FUNCTION_BLOCK FB_WP_Ablaufsteuerung
VAR_IN_OUT
	Zustand			: ST_WP_Zustand;
	Stellwert		: ST_WP_Stellwert;
END_VAR
VAR_INPUT
	Steuerung		: ST_WP_Steuerung;
	Parameter		: ST_WP_Parameter;
END_VAR
VAR_OUTPUT
END_VAR
VAR
	Timer			: TON;
END_VAR

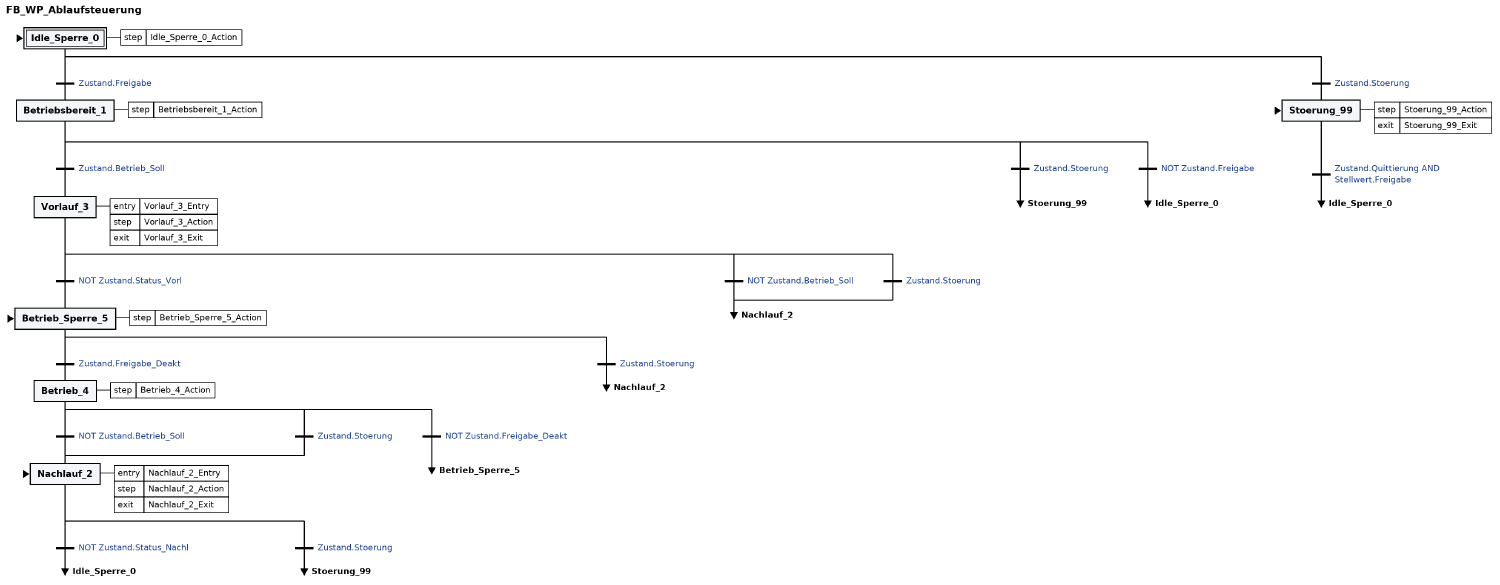
INITIAL_STEP Idle_Sperre_0:
    Idle_Sperre_0_Action(N);  // step action
END_STEP
TRANSITION FROM Idle_Sperre_0 TO Betriebsbereit_1
    := Zustand.Freigabe;
END_TRANSITION
TRANSITION FROM Idle_Sperre_0 TO Stoerung_99
    := Zustand.Stoerung;
END_TRANSITION
STEP Stoerung_99:
    Stoerung_99_Action(N);  // step action
    Stoerung_99_Exit(P0);  // exit action
END_STEP
TRANSITION FROM Stoerung_99 TO Idle_Sperre_0
    := Zustand.Quittierung AND Stellwert.Freigabe;
END_TRANSITION
STEP Betriebsbereit_1:
    Betriebsbereit_1_Action(N);  // step action
END_STEP
TRANSITION FROM Betriebsbereit_1 TO Vorlauf_3
    := Zustand.Betrieb_Soll;
END_TRANSITION
TRANSITION FROM Betriebsbereit_1 TO Stoerung_99
    := Zustand.Stoerung;
END_TRANSITION
TRANSITION FROM Betriebsbereit_1 TO Idle_Sperre_0
    := NOT Zustand.Freigabe;
END_TRANSITION
STEP Vorlauf_3:
    Vorlauf_3_Entry(P1);  // entry action
    Vorlauf_3_Action(N);  // step action
    Vorlauf_3_Exit(P0);  // exit action
END_STEP
TRANSITION FROM Vorlauf_3 TO Betrieb_Sperre_5
    := NOT Zustand.Status_Vorl;
END_TRANSITION
TRANSITION FROM Vorlauf_3 TO Nachlauf_2
    := NOT Zustand.Betrieb_Soll;
END_TRANSITION
TRANSITION FROM Vorlauf_3 TO Nachlauf_2
    := Zustand.Stoerung;
END_TRANSITION
STEP Betrieb_Sperre_5:
    Betrieb_Sperre_5_Action(N);  // step action
END_STEP
TRANSITION FROM Betrieb_Sperre_5 TO Betrieb_4
    := Zustand.Freigabe_Deakt;
END_TRANSITION
TRANSITION FROM Betrieb_Sperre_5 TO Nachlauf_2
    := Zustand.Stoerung;
END_TRANSITION
STEP Betrieb_4:
    Betrieb_4_Action(N);  // step action
END_STEP
TRANSITION FROM Betrieb_4 TO Nachlauf_2
    := NOT Zustand.Betrieb_Soll;
END_TRANSITION
TRANSITION FROM Betrieb_4 TO Nachlauf_2
    := Zustand.Stoerung;
END_TRANSITION
TRANSITION FROM Betrieb_4 TO Betrieb_Sperre_5
    := NOT Zustand.Freigabe_Deakt;
END_TRANSITION
STEP Nachlauf_2:
    Nachlauf_2_Entry(P1);  // entry action
    Nachlauf_2_Action(N);  // step action
    Nachlauf_2_Exit(P0);  // exit action
END_STEP
TRANSITION FROM Nachlauf_2 TO Idle_Sperre_0
    := NOT Zustand.Status_Nachl;
END_TRANSITION
TRANSITION FROM Nachlauf_2 TO Stoerung_99
    := Zustand.Stoerung;
END_TRANSITION

ACTION Betrieb_4_Action:
(* Stellwert setzen *)
Stellwert.Betrieb := TRUE;

(* Zustand setzen *)
Zustand.Status := E_WP_Zustand_Status_Betrieb;
END_ACTION

ACTION Betrieb_Sperre_5_Action:
(* Stellwert setzen *)
Stellwert.Betrieb := TRUE;

(* Zustand setzen *)
Zustand.Status := E_WP_Zustand_Status_Betrieb_Sperre;
END_ACTION

ACTION Betriebsbereit_1_Action:
(* Stellwert setzen *)
Stellwert.Betrieb := FALSE;
Stellwert.Freigabe := TRUE;

(* Zustand setzen *)
Zustand.Status := E_WP_Zustand_Status_Betriebsbereit;
END_ACTION

ACTION Idle_Sperre_0_Action:
(* Stellwert setzen *)
Stellwert.Betrieb := FALSE;

(* Zustand setzen *)
Zustand.Status := E_WP_Zustand_Status_Idle_Sperre;
END_ACTION

ACTION Nachlauf_2_Action:
(* Nachlauf Timer starten *)
Timer( 	IN := Zustand.Status_Nachl,
		PT := DINT_TO_TIME(Parameter.Zeit_Nachl)
);
Zustand.Status_Nachl	:= NOT(Timer.Q AND NOT Zustand.Betrieb);

(* Stellwert setzen *)
Stellwert.Betrieb := FALSE;
Stellwert.Freigabe := FALSE;

(* Zustand setzen *)
Zustand.Status := E_WP_Zustand_Status_Nachl;
END_ACTION

ACTION Nachlauf_2_Entry:
Zustand.Status_Nachl := TRUE;
(* Reset Timer *)
Timer(IN := FALSE);
END_ACTION

ACTION Nachlauf_2_Exit:
Zustand.Status_Nachl := FALSE;
END_ACTION

ACTION Stoerung_99_Action:
(* Stellwert setzen *)
Stellwert.Betrieb := FALSE;

(* Zustand setzen *)
Zustand.Stoerung := TRUE;
Zustand.Status := E_WP_Zustand_Status_Stoerung;
END_ACTION

ACTION Stoerung_99_Exit:
Zustand.Stoerung	:= FALSE;
END_ACTION

ACTION Vorlauf_3_Action:
(* Vorlaufzeit Timer starten *)
Timer( 	IN := Zustand.Status_Vorl,
		PT := DINT_TO_TIME(Parameter.Zeit_Vorl)
);
Zustand.Status_Vorl := NOT (Timer.Q);

(* Stellwert setzen *)
IF Stellwert.Freigabe THEN
	Stellwert.Betrieb := TRUE;
END_IF

(* Zustand setzen *)
Zustand.Status := E_WP_Zustand_Status_Vorl;
END_ACTION

ACTION Vorlauf_3_Entry:
Zustand.Status_Vorl := TRUE;
(* Reset Timer *)
Timer(IN := FALSE);
END_ACTION

ACTION Vorlauf_3_Exit:
Zustand.Status_Vorl := FALSE;
END_ACTION

END_FUNCTION_BLOCK

(* stored: Version 1.1.0.1, ProductVersion 3.1.4024.9
   POU FB_WP_Ablaufsteuerung: Id {dd15999f-292f-4a8b-9368-8693d9b7681d}, SpecialFunc None
   Action Betrieb_4_Action: Id {6256f494-f51c-448d-819e-5fdb742b51a2}
   Action Betrieb_Sperre_5_Action: Id {c69565df-6e9c-4316-80ba-343bd7669a1a}
   Action Betriebsbereit_1_Action: Id {86ac766d-643a-4a88-a5e4-ba51f6d7a02e}
   Action Idle_Sperre_0_Action: Id {00132048-9c42-4c5d-b2b4-ad78d6e949bb}
   Action Nachlauf_2_Action: Id {9d773eb8-15ed-4d2c-b4d7-48bf162be89a}
   Action Nachlauf_2_Entry: Id {9269b023-829f-474a-ac16-5b1ffe57039b}
   Action Nachlauf_2_Exit: Id {0d3df664-91ca-43f3-89ea-26784278a22e}
   Action Stoerung_99_Action: Id {0c2f8b67-78a2-41d0-a4fa-4f845480bb23}
   Action Stoerung_99_Exit: Id {6c25e45e-b0f9-4c0e-9902-62e0f04c3116}
   Action Vorlauf_3_Action: Id {97068a46-a71d-4934-b5a6-929ee3af662a}
   Action Vorlauf_3_Entry: Id {6a20d783-b139-4a0a-a788-9aed4489752e}
   Action Vorlauf_3_Exit: Id {ed87d5de-7c08-4a4d-915b-8e36a1f8528c} *)
